{attribute addProperty BoxType "EK1100-0000-0018"}
{attribute addProperty Id "Beckhoff_EL6xxxEK1122Beckhoff_EL6xxxEK1122_C6B70D18162A_0001_EL6001_0000_0000EL6001_A7B322AF48060A_0002_EL6001_0000_0016EL6001_1A54FD5351564.375A_0003_EL6001_0000_0017EL6001_5D31AA5148060A_0004_EL6001_0000_0018EL6001_5D31AA5148060A_0005_EL6001_0000_0019EL6001_5D31AA5148060A_0006_EL6001_0000_0020EL6001_5D31AA5148060A_0007_EL6002_0000_0016EL6002_55A24E9B934116.75A_0008_EL6002_0000_0017EL6002_45B1C254864108A_0009_EL6002_0000_0018EL6002_45B1C254864108A_0010_EL6002_0000_0019EL6002_45B1C254864108A_0011_EL6021_0000_0000EL6021_A7B322AF48060A_0012_EL6021_0000_0016EL6021_1A54FD5351564.375A_0013_EL6021_0000_0017EL6021_1A54FD5351564.375A_0014_EL6021_0000_0018EL6021_2B16659A48060A_0015_EL6021_0000_0019EL6021_2B16659A48060A_0016_EL6021_0000_0020EL6021_2B16659A48060A_0017_EL6021_0000_0021EL6021_2B16659A48060A_0018_EL6021_0021_0018EL6021_2B16659A48060A_0019_EL6021_0021_0019EL6021_2B16659A48060A_0020_EL6021_0021_0020EL6021_2B16659A48060A_0021_EL6021_0021_0021EL6021_2B16659A48060A_0022_EL6022_0000_0016EL6022_55A24E9B934116.75A_0023_EL6022_0000_0017EL6022_55A24E9B934116.75A_0024_EL6022_0000_0018EL6022_55A24E9B934116.75A_0025_EL6022_0000_0019EL6022_A0C112E7864108A_0026_EL6070_0000_0016EL6070_194A340D8010A_0027_EL6070_0000_0017EL6070_194A340D8010A_0028_EL6070_0000_0018EL6070_194A340D8010A_0029_EL6070_0000_0019EL6070_194A340D8010A_0030_EL6070_0033_0016EL6070_194A340D8010A_0031_EL6070_0033_0017EL6070_194A340D8010A_0032_EL6070_0033_0018EL6070_194A340D8010A_0033_EL6070_0033_0019EL6070_194A340D8010A_0034_EL6080_0000_0016EL6080_49EF2FC49612A_0035_EL6080_0000_0017EL6080_49EF2FC49612A_0036_EL6080_0000_0018EL6080_820BDBFD12816A_0037_EL6080_0000_0020EL6080_820BDBFD12816A_0038_EL6090_0000_0016EL6090_C46C03A814418A_0039_EL6090_0000_0017EL6090_C46C03A814418A_0040_EL6201_0000_0017EL6201_34DED8B972090A_0041_EL6201_0000_0018EL6201_C873A9DB75294A_0042_EL6201_0000_0019EL6201_C873A9DB75294A_0043_EL6224_0000_0016EL6224_CC9621B717622A_0044_EL6224_0000_0017EL6224_7C2B6CA219224A_0045_EL6224_0000_0018EL6224_7C2B6CA219224A_0046_EL6224_0000_0019EL6224_7C2B6CA219224A_0047_EL6224_0000_0020EL6224_7C2B6CA219224A_0048_EL6224_0000_0021EL6224_7C2B6CA219224A_0049_EL6224_0090_0016EL6224_193A140119224A_0050_EL6224_0090_0017EL6224_193A140119224"}
{attribute addProperty CRC "3702620105"}
{attribute addProperty SizeInBites "20593"}
{attribute addProperty SizeInBytes "2574.125"}
TYPE Beckhoff_EL6xxx_DCB17FC9 EXTENDS EK1100_179A0949 :
STRUCT
	{attribute addProperty Name "Beckhoff_EL6xxxEK1122"}
	Beckhoff_EL6xxxEK1122 : Beckhoff_EL6xxxEK1122_C6B70D18;
	{attribute addProperty Name "A_0001_EL6001_0000_0000"}
	A_0001_EL6001_0000_0000 : EL6001_A7B322AF;
	{attribute addProperty Name "A_0002_EL6001_0000_0016"}
	A_0002_EL6001_0000_0016 : EL6001_1A54FD53;
	{attribute addProperty Name "A_0003_EL6001_0000_0017"}
	A_0003_EL6001_0000_0017 : EL6001_5D31AA51;
	{attribute addProperty Name "A_0004_EL6001_0000_0018"}
	A_0004_EL6001_0000_0018 : EL6001_5D31AA51;
	{attribute addProperty Name "A_0005_EL6001_0000_0019"}
	A_0005_EL6001_0000_0019 : EL6001_5D31AA51;
	{attribute addProperty Name "A_0006_EL6001_0000_0020"}
	A_0006_EL6001_0000_0020 : EL6001_5D31AA51;
	{attribute addProperty Name "A_0007_EL6002_0000_0016"}
	A_0007_EL6002_0000_0016 : EL6002_55A24E9B;
	{attribute addProperty Name "A_0008_EL6002_0000_0017"}
	A_0008_EL6002_0000_0017 : EL6002_45B1C254;
	{attribute addProperty Name "A_0009_EL6002_0000_0018"}
	A_0009_EL6002_0000_0018 : EL6002_45B1C254;
	{attribute addProperty Name "A_0010_EL6002_0000_0019"}
	A_0010_EL6002_0000_0019 : EL6002_45B1C254;
	{attribute addProperty Name "A_0011_EL6021_0000_0000"}
	A_0011_EL6021_0000_0000 : EL6021_A7B322AF;
	{attribute addProperty Name "A_0012_EL6021_0000_0016"}
	A_0012_EL6021_0000_0016 : EL6021_1A54FD53;
	{attribute addProperty Name "A_0013_EL6021_0000_0017"}
	A_0013_EL6021_0000_0017 : EL6021_1A54FD53;
	{attribute addProperty Name "A_0014_EL6021_0000_0018"}
	A_0014_EL6021_0000_0018 : EL6021_2B16659A;
	{attribute addProperty Name "A_0015_EL6021_0000_0019"}
	A_0015_EL6021_0000_0019 : EL6021_2B16659A;
	{attribute addProperty Name "A_0016_EL6021_0000_0020"}
	A_0016_EL6021_0000_0020 : EL6021_2B16659A;
	{attribute addProperty Name "A_0017_EL6021_0000_0021"}
	A_0017_EL6021_0000_0021 : EL6021_2B16659A;
	{attribute addProperty Name "A_0018_EL6021_0021_0018"}
	A_0018_EL6021_0021_0018 : EL6021_2B16659A;
	{attribute addProperty Name "A_0019_EL6021_0021_0019"}
	A_0019_EL6021_0021_0019 : EL6021_2B16659A;
	{attribute addProperty Name "A_0020_EL6021_0021_0020"}
	A_0020_EL6021_0021_0020 : EL6021_2B16659A;
	{attribute addProperty Name "A_0021_EL6021_0021_0021"}
	A_0021_EL6021_0021_0021 : EL6021_2B16659A;
	{attribute addProperty Name "A_0022_EL6022_0000_0016"}
	A_0022_EL6022_0000_0016 : EL6022_55A24E9B;
	{attribute addProperty Name "A_0023_EL6022_0000_0017"}
	A_0023_EL6022_0000_0017 : EL6022_55A24E9B;
	{attribute addProperty Name "A_0024_EL6022_0000_0018"}
	A_0024_EL6022_0000_0018 : EL6022_55A24E9B;
	{attribute addProperty Name "A_0025_EL6022_0000_0019"}
	A_0025_EL6022_0000_0019 : EL6022_A0C112E7;
	{attribute addProperty Name "A_0026_EL6070_0000_0016"}
	A_0026_EL6070_0000_0016 : EL6070_194A340D;
	{attribute addProperty Name "A_0027_EL6070_0000_0017"}
	A_0027_EL6070_0000_0017 : EL6070_194A340D;
	{attribute addProperty Name "A_0028_EL6070_0000_0018"}
	A_0028_EL6070_0000_0018 : EL6070_194A340D;
	{attribute addProperty Name "A_0029_EL6070_0000_0019"}
	A_0029_EL6070_0000_0019 : EL6070_194A340D;
	{attribute addProperty Name "A_0030_EL6070_0033_0016"}
	A_0030_EL6070_0033_0016 : EL6070_194A340D;
	{attribute addProperty Name "A_0031_EL6070_0033_0017"}
	A_0031_EL6070_0033_0017 : EL6070_194A340D;
	{attribute addProperty Name "A_0032_EL6070_0033_0018"}
	A_0032_EL6070_0033_0018 : EL6070_194A340D;
	{attribute addProperty Name "A_0033_EL6070_0033_0019"}
	A_0033_EL6070_0033_0019 : EL6070_194A340D;
	{attribute addProperty Name "A_0034_EL6080_0000_0016"}
	A_0034_EL6080_0000_0016 : EL6080_49EF2FC4;
	{attribute addProperty Name "A_0035_EL6080_0000_0017"}
	A_0035_EL6080_0000_0017 : EL6080_49EF2FC4;
	{attribute addProperty Name "A_0036_EL6080_0000_0018"}
	A_0036_EL6080_0000_0018 : EL6080_820BDBFD;
	{attribute addProperty Name "A_0037_EL6080_0000_0020"}
	A_0037_EL6080_0000_0020 : EL6080_820BDBFD;
	{attribute addProperty Name "A_0038_EL6090_0000_0016"}
	A_0038_EL6090_0000_0016 : EL6090_C46C03A8;
	{attribute addProperty Name "A_0039_EL6090_0000_0017"}
	A_0039_EL6090_0000_0017 : EL6090_C46C03A8;
	{attribute addProperty Name "A_0040_EL6201_0000_0017"}
	A_0040_EL6201_0000_0017 : EL6201_34DED8B9;
	{attribute addProperty Name "A_0041_EL6201_0000_0018"}
	A_0041_EL6201_0000_0018 : EL6201_C873A9DB;
	{attribute addProperty Name "A_0042_EL6201_0000_0019"}
	A_0042_EL6201_0000_0019 : EL6201_C873A9DB;
	{attribute addProperty Name "A_0043_EL6224_0000_0016"}
	A_0043_EL6224_0000_0016 : EL6224_CC9621B7;
	{attribute addProperty Name "A_0044_EL6224_0000_0017"}
	A_0044_EL6224_0000_0017 : EL6224_7C2B6CA2;
	{attribute addProperty Name "A_0045_EL6224_0000_0018"}
	A_0045_EL6224_0000_0018 : EL6224_7C2B6CA2;
	{attribute addProperty Name "A_0046_EL6224_0000_0019"}
	A_0046_EL6224_0000_0019 : EL6224_7C2B6CA2;
	{attribute addProperty Name "A_0047_EL6224_0000_0020"}
	A_0047_EL6224_0000_0020 : EL6224_7C2B6CA2;
	{attribute addProperty Name "A_0048_EL6224_0000_0021"}
	A_0048_EL6224_0000_0021 : EL6224_7C2B6CA2;
	{attribute addProperty Name "A_0049_EL6224_0090_0016"}
	A_0049_EL6224_0090_0016 : EL6224_193A1401;
	{attribute addProperty Name "A_0050_EL6224_0090_0017"}
	A_0050_EL6224_0090_0017 : EL6224_193A1401;
END_STRUCT
END_TYPE

(* stored: Version 1.2.0.0, ProductVersion 3.1.4024.9
   DUT Beckhoff_EL6xxx_DCB17FC9: Id {f04c0dfc-1460-4ade-8c0f-be3a908eefa3} *)
